# EPICS substitutions: OLD/mc14/tpmacApp/Db/motor.substitutions
file "db/motor.db"
{
pattern
{P,              M,                     MOTOR,  PORT,  ADDR,  DESC,        DTYP,      MRES,   EGU,  PREC,  ALIAS }
{"XF:23ID2-ES",  "{APPES:1-Ax:X}Mtr",  "M0",   "P0",  1,     "APPES X",    asynMotor, 3.294063E-5,  "mm", 3,     ""    }
{"XF:23ID2-ES",  "{APPES:1-Ax:Y}Mtr",  "M0",   "P0",  2,     "APPES Y",    asynMotor, 1.984375E-4,  "mm", 3,     ""    }
{"XF:23ID2-ES",  "{APPES:1-Ax:Z}Mtr",  "M0",   "P0",  3,     "APPES Z",    asynMotor, 3.294063E-5,  "mm", 3,     ""    }
{"XF:23ID2-ES",  "{APPES:1-Ax:R}Mtr",  "M0",   "P0",  4,     "APPES R",    asynMotor, 5.625000E-4,  "deg", 3,     ""    }
}
